Staubli VAL3: PointGrey.pjx

Parameters version=s7.6.2 stackSize=5000 millimeterUnit=true
Program file=create.pgx
Program file=detection.pgx
Program file=getMaxNumOfPart.pgx
Program file=getObjectData.pgx
Program file=getObjectLatch.pgx
Program file=getValue.pgx
Program file=init.pgx
Program file=initvis.pgx
Program file=isDetected.pgx
Program file=kill.pgx
Program file=resetTask.pgx
Program file=sortObjects.pgx
Program file=start.pgx
Program file=stop.pgx
Data file=PointGrey.dtx
Library alias=ut path=Disk://Tracking/Tools/util/util.pjx autoload=true password=
Library alias=sck path=Disk://Tracking/io/sockets/sockets.pjx autoload=true password=
Type name=object path=Disk://Tracking/Templates/object/object.pjx
